ABB RobotStudio station: mine.rsstn

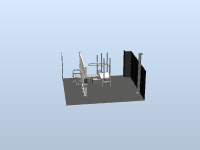
Station Station (saved by RobotStudio format 5)
Layout (positions relative to the parent item):
  - IRB120_3_58__01 [mechanism, from Robots\IRB120_3_58_G_01.rslib] at (0, 0, 0) mm; joint values [0, 0, 0.7854, 0, 0, 0] (rad or m)
  - MyNewTool [mechanism] at (250, 0, 308.5) mm, rotated rx -90 ry 0 rz 180 deg
      TCP SuctionCup at (0, 65, 0) mm
      links: End Effector
  - Robot Cell - Base-1 [part] at (-2877, -3695.5, -586) mm
  - Robot Cell - Cell Barrier-1 [part] at (-2877, -3695.5, -586) mm
  - Robot Cell - Converyer Enclosure-1 [part] at (-2877, -3695.5, -586) mm
  - Robot Cell - Conveyer-2 [part] at (-2877, -3695.5, -586) mm
  - Robot Cell - E-Stop and Motor On Mounting Plate-1 [part] at (-2877, -3695.5, -586) mm
  - Robot Cell - E-Stop Master-1 [part] at (-2877, -3695.5, -586) mm
  - Robot Cell - Floor-1 [part] at (-2877, -3695.5, -586) mm
  - Robot Cell - Hazard Frame Member-1 [part] at (-2877, -3695.5, -586) mm
  - Robot Cell - Intermediate Table Frame Members-1 [part] at (-2877, -3695.5, -586) mm
  - Robot Cell - Intermediate Table Frame Members-2 [part] at (-2877, -3695.5, -586) mm
  - Robot Cell - Large Frame Member-1 [part] at (-2877, -3695.5, -586) mm
  - Robot Cell - Large Frame Member-2 [part] at (-2877, -3695.5, -586) mm
  - Robot Cell - Large Frame Member-3 [part] at (-2877, -3695.5, -586) mm
  - Robot Cell - Large Frame Member-6 [part] at (-2877, -3695.5, -586) mm
  - Robot Cell - Large Frame Member-7 [part] at (-2877, -3695.5, -586) mm
  - Robot Cell - Large Frame Member-8 [part] at (-2877, -3695.5, -586) mm
  - Robot Cell - Large Frame Member-9 [part] at (-2877, -3695.5, -586) mm
  - Robot Cell - Large Frame Member-10 [part] at (-2877, -3695.5, -586) mm
  - Robot Cell - Large Remote E-Stop-1 [part] at (-2877, -3695.5, -586) mm
  - Robot Cell - Motor Panel-1 [part] at (-2877, -3695.5, -586) mm
  - Robot Cell - Robot Cell Bar-1 [part] at (-2877, -3695.5, -586) mm
  - Robot Cell - Robot Motor Controller-1 [part] at (-2877, -3695.5, -586) mm
  - Robot Cell - Small Frame Member-1 [part] at (-2877, -3695.5, -586) mm
  - Robot Cell - Small Remote E-Stop-1 [part] at (-2877, -3695.5, -586) mm
  - Robot Cell - Small Remote E-Stop-2 [part] at (-2877, -3695.5, -586) mm
  - Robot Cell - Table Base Frame Member-1 [part] at (-2877, -3695.5, -586) mm
  - Robot Cell - Table Base Frame Member-2 [part] at (-2877, -3695.5, -586) mm
  - Robot Cell - Table-1 [part] at (-2877, -3695.5, -586) mm
  - Conveyor Frame [frame] at (-300, 409, 22) mm
  - T1 [frame] at (175, 0, 147) mm
  - T2 [frame] at (175, -520, 147) mm
  - T3 [frame] at (175, 520, 147) mm
  - T4 [frame] at (548.6, 0, 147) mm
